# EPICS autosave request: iocs/meascomp/usb-ctr-ioc/auto_settings.req
# Settings restored at the next start of usb-ctr-ioc.
# Ported from upstream USBCTR_settings.req and the per-template
# measComp*_settings.req files it includes.
#
# Macros: P (record prefix)

$(P)PollSleepMS

$(P)Bd1
$(P)Bd2
$(P)Bd3
$(P)Bd4
$(P)Bd5
$(P)Bd6
$(P)Bd7
$(P)Bd8

$(P)PulseGen1Period
$(P)PulseGen1Width
$(P)PulseGen1Delay
$(P)PulseGen1Count
$(P)PulseGen1IdleState
$(P)PulseGen2Period
$(P)PulseGen2Width
$(P)PulseGen2Delay
$(P)PulseGen2Count
$(P)PulseGen2IdleState
$(P)PulseGen3Period
$(P)PulseGen3Width
$(P)PulseGen3Delay
$(P)PulseGen3Count
$(P)PulseGen3IdleState
$(P)PulseGen4Period
$(P)PulseGen4Width
$(P)PulseGen4Delay
$(P)PulseGen4Count
$(P)PulseGen4IdleState

$(P)MCS:PresetReal
$(P)MCS:Dwell
$(P)MCS:Prescale
$(P)MCS:PrescaleCounter
$(P)MCS:Point0Action
$(P)MCS:ChannelAdvance
$(P)MCS:TrigMode
$(P)MCS:NuseAll
$(P)MCS:MCSCounter1Enable
$(P)MCS:MCSCounter2Enable
$(P)MCS:MCSCounter3Enable
$(P)MCS:MCSCounter4Enable
$(P)MCS:MCSCounter5Enable
$(P)MCS:MCSCounter6Enable
$(P)MCS:MCSCounter7Enable
$(P)MCS:MCSCounter8Enable
$(P)MCS:MCSDIOEnable
$(P)MCS:EnableClientWait
$(P)MCS:ReadAll.SCAN

$(P)scaler1.TP
$(P)scaler1.FREQ
